// TwinCAT 3 PLC project PLC_851
// ProgramVersion: 3.1.4024.0
// libraries:
//   Tc2_Standard, * (Beckhoff Automation GmbH)
//   Tc2_System, * (Beckhoff Automation GmbH)
//   Tc3_Module, * (Beckhoff Automation GmbH)
// project tree:
//   DUTs/ E_TL_Phase.TcDUT
//   / GlobalTextList.TcGTLO, PlcTask.TcTTO, Visualisierungsmanager.TcVMO (not stored)
//   GVLs/ GVL_HMI_TrafficLight.TcGVL
//   POUs/ FB_TrafficLight_ENUM.TcPOU, FB_TrafficLight_STP.TcPOU, MAIN.TcPOU
//   POUs/TOOLS/ FB_Toggle.TcPOU
//   VISUs/ TrafficLight.TcVIS
// real-time tasks:
//   TASK PlcTask: cycle T#10ms, priority 20, ADS port 350

CONFIGURATION PLC_851
    RESOURCE PLC ON TwinCAT3
        TASK PlcTask(INTERVAL := T#10ms, PRIORITY := 20);
        PROGRAM MAIN WITH PlcTask : MAIN;
    END_RESOURCE
END_CONFIGURATION

// ---- DUTs/E_TL_Phase.TcDUT
{attribute 'qualified_only'}
{attribute 'strict'}
TYPE E_TL_Phase :
(
	INIT := 0,
	RED,		//1
	GREEN,		//2
	YELLOW,		//3 
	YELLOWRED	//4
);
END_TYPE

// ---- GVLs/GVL_HMI_TrafficLight.TcGVL
VAR_GLOBAL
	// Ampel 1
	LED_Red			: BOOL;
	LED_Yellow		: BOOL;
	LED_Green		: BOOL;
	
	btnReset		: BOOL;
	btnActive		: BOOL;
	
	// Ampel 2
	LED_Red_1		: BOOL;
	LED_Yellow_1	: BOOL;
	LED_Green_1		: BOOL;
	
	btnReset_1		: BOOL;
	btnActive_1		: BOOL;
	
	bBlink			: BOOL;

END_VAR

// ---- POUs/MAIN.TcPOU
PROGRAM MAIN
VAR
	fbTakt	: FB_Toggle;
	fbTrafficLight_enum	: FB_TrafficLight_ENUM;
	fbTrafficLight_stp	: FB_TrafficLight_STP;
END_VAR

fbTakt();
fbTrafficLight_enum();
fbTrafficLight_stp();

END_PROGRAM

// ---- POUs/TOOLS/FB_Toggle.TcPOU
FUNCTION_BLOCK FB_Toggle
VAR_INPUT
END_VAR
VAR_OUTPUT
END_VAR
VAR
	Timer_1s 	: TON; 		// Timer für den Takt
	Timer_500ms	: TON;		// Timer für Ampelblinktakt
	Cycle_1s	: BOOL;		// Tooglevariable
END_VAR

// Timmer 1s Zyklus
Timer_1s(IN:=NOT Timer_1s.Q ,
		 PT:=T#1S );
		 
Cycle_1s := Cycle_1s XOR Timer_1s.Q;

//Timer für Ampelblinktakt
Timer_500ms(IN:=NOT Timer_500ms.Q ,
		 	PT:=T#600MS );
			
bBlink := bBlink XOR Timer_500ms.Q;

END_FUNCTION_BLOCK

// ---- POUs/FB_TrafficLight_ENUM.TcPOU
FUNCTION_BLOCK FB_TrafficLight_ENUM
VAR_INPUT
END_VAR
VAR_OUTPUT
END_VAR
VAR
	state		: INT;
	tRed		: TON;		// Leuchtdauer Rot
	tRedYellow	: TON;	 	// Leuchtdauer RotGelb
	tGreen		: TON;		// Leuchtaduer Gruen
	tYellow		: TON;		// Leuchtdauer Gelb
END_VAR

CASE state OF
	E_TL_Phase.INIT:
			LED_Red	:= FALSE;
			LED_Yellow := bBlink;
			LED_Green := FALSE;
	
	E_TL_Phase.RED:
			LED_Red	:= TRUE;
			LED_Yellow := FALSE;
			LED_Green := FALSE;
			IF tRed.Q THEN
				state := E_TL_Phase.YELLOWRED;
			END_IF
			
	E_TL_Phase.YELLOWRED:
			LED_Red	:= TRUE;
			LED_Yellow := TRUE;
			LED_Green := FALSE;
			IF tRedYellow.Q THEN
				state := E_TL_Phase.GREEN;
			END_IF
			
	E_TL_Phase.GREEN:
			LED_Red	:= FALSE;
			LED_Yellow := FALSE;
			LED_Green := TRUE;
			IF tGreen.Q THEN
				state :=E_TL_Phase.YELLOW;
			END_IF
			
	E_TL_Phase.YELLOW:
			LED_Red	:= FALSE;
			LED_Yellow := TRUE;
			LED_Green := FALSE;
			IF tYellow.Q THEN
				state := E_TL_Phase.RED;
			END_IF
ELSE
			LED_Yellow := bBlink;
			LED_Red	:= FALSE;
			LED_Green := FALSE;
END_CASE

IF btnReset THEN
	state := E_TL_Phase.INIT;
	ELSE ;
END_IF

IF btnActive AND (state = 0) THEN
	state := E_TL_Phase.RED;
END_IF


// Timer

tRed(	IN:=(state =  E_TL_Phase.RED),
		PT := T#2S);
		
tRedYellow(	IN:=(state =  E_TL_Phase.YELLOWRED),
		PT := T#2S);
		
tGreen(	IN:=(state =  E_TL_Phase.GREEN),
		PT := T#2S);

tYellow(	IN:=(state =  E_TL_Phase.YELLOW),
		PT := T#2S);

END_FUNCTION_BLOCK

// ---- POUs/FB_TrafficLight_STP.TcPOU
FUNCTION_BLOCK FB_TrafficLight_STP
VAR_INPUT
END_VAR
VAR_OUTPUT
END_VAR
VAR
	iStep		: INT;		// Schrittnummer
	tRed		: TON;		// Leuchtdauer Rot
	tRedYellow	: TON;	 	// Leuchtdauer RotGelb
	tGreen		: TON;		// Leuchtaduer Gruen
	tYellow		: TON;		// Leuchtdauer Gelb

END_VAR

CASE iStep OF
	0:	// INIT
			LED_Red	:= FALSE;
			LED_Yellow := bBlink;
			LED_Green := FALSE;
	
	1:	// RED
			LED_Red	:= TRUE;
			LED_Yellow := FALSE;
			LED_Green := FALSE;
			IF tRed.Q THEN
				iStep := E_TL_Phase.YELLOWRED;
			END_IF
			
	2:	// YELLOWRED
			LED_Red	:= TRUE;
			LED_Yellow := TRUE;
			LED_Green := FALSE;
			IF tRedYellow.Q THEN
				iStep := E_TL_Phase.GREEN;
			END_IF
			
	3:	// GREEN
			LED_Red	:= FALSE;
			LED_Yellow := FALSE;
			LED_Green := TRUE;
			IF tGreen.Q THEN
				iStep :=E_TL_Phase.YELLOW;
			END_IF
			
	4:	// YELLOW
			LED_Red	:= FALSE;
			LED_Yellow := TRUE;
			LED_Green := FALSE;
			IF tYellow.Q THEN
				iStep := E_TL_Phase.RED;
			END_IF
ELSE
			LED_Yellow := bBlink;
			LED_Red	:= FALSE;
			LED_Green := FALSE;
END_CASE

IF btnReset THEN
	iStep := E_TL_Phase.INIT;
	ELSE ;
END_IF

IF btnActive AND (iStep = 0) THEN
	iStep := E_TL_Phase.RED;
END_IF


// Timer

tRed(		IN:=(iStep = 1),
			PT := T#2S);
		
tRedYellow(	IN:=(iStep = 2),
			PT := T#2S);
		
tGreen(		IN:=(iStep = 3),
			PT := T#2S);

tYellow(	IN:=(iStep = 4),
			PT := T#2S);

END_FUNCTION_BLOCK

// ---- GlobalTextList.TcGTLO
TEXTLIST GlobalTextList
  58 = 'Active'
  712 = 'Ampel ENUM'
  851 = 'Ampel STP'
  547 = 'ENUM'
  194 = 'Reset'
  840 = 'STP'
END_TEXTLIST

// ---- VISUs/TrafficLight.TcVIS
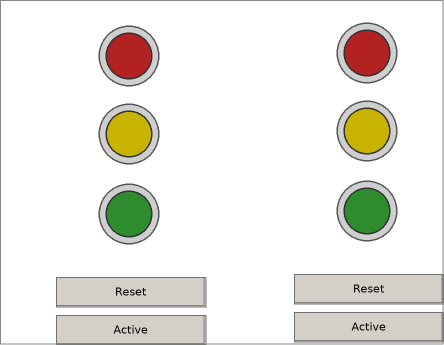
VISUALIZATION TrafficLight  // 444x345
    Lamp1 (94,21 70x70), variable: GVL_HMI_TrafficLight.LED_Red, style: Lamp-Lamp1-Red
    Lamp1 (94,99 70x70), variable: GVL_HMI_TrafficLight.LED_Yellow, style: Lamp-Lamp1-Yellow
    Lamp1 (94,179 70x70), variable: GVL_HMI_TrafficLight.LED_Green, style: Lamp-Lamp1-Green
    Button (56,277 150x30), "Reset"
        tap GVL_HMI_TrafficLight.btnReset
    Button (56,315 150x30), "Active"
        tap GVL_HMI_TrafficLight.btnActive
    Lamp1 (332,18 70x70), variable: GVL_HMI_TrafficLight.LED_Red_1, style: Lamp-Lamp1-Red
    Lamp1 (332,96 70x70), variable: GVL_HMI_TrafficLight.LED_Yellow_1, style: Lamp-Lamp1-Yellow
    Lamp1 (332,176 70x70), variable: GVL_HMI_TrafficLight.LED_Green_1, style: Lamp-Lamp1-Green
    Button (294,274 150x30), "Reset"
        tap GVL_HMI_TrafficLight.btnReset_1
    Button (294,312 150x30), "Active"
        tap GVL_HMI_TrafficLight.btnActive_1
END_VISUALIZATION
